FUNCTION_BLOCK A24 EXTENDS GenericSubarea

SUPER^();

METHOD PROTECTED callHardware : BOOL
VAR_INPUT
END_VAR
END_METHOD

METHOD PROTECTED runModules : BOOL
VAR_INPUT
END_VAR
// NETWORK 1
END_METHOD

METHOD PROTECTED setupHardware : BOOL
VAR
	i : INT;
END_VAR
END_METHOD

END_FUNCTION_BLOCK

(* stored: Version 1.1.0.1, ProductVersion 3.1.4024.11
   POU A24: Id {9825abd9-77b4-48ca-9d54-54afdff6fff9}, SpecialFunc None
   Method callHardware: Id {c8ac936c-7d12-438b-a0a6-3c27a72b6d3c}
   Method runModules: Id {2010770a-d99d-45d5-a371-a2a4fae79adb}
   Method setupHardware: Id {4c5ab590-4716-4e6c-afb0-86b3c85cecc7} *)
